(* IEC 61131-3 sources: AutomationStudio/BramaWjazdowa, 3 files *)

(* ---- Types.typ ---- *)
TYPE
	OperatorTyp : STRUCT
		diStart : BOOL;
		diStop : BOOL:= TRUE;
		diEStop : BOOL := TRUE;
		diKasujAwaria: BOOL; (*Przycisk kasowania awarii*)
		doSystemAktywny: BOOL; (*Lampka systemu aktywny*)
		doAwaria : BOOL; (*Lampka Awaria*)
		diGateOpen : BOOL;
		diGateClose : BOOL;
		Pilot : PilotTyp;
	END_STRUCT;

	PilotTyp : STRUCT
		diGateOpen : BOOL;
		diGateClose : BOOL;
		diEStop : BOOL := TRUE;
	END_STRUCT;

	GateTyp : STRUCT
		diSafetySensor : BOOL := TRUE;
		diGateClosed : BOOL:= TRUE;
		diGateOpened : BOOL:= TRUE;
		diTemperature : BOOL := TRUE;
		doOpenGate : BOOL;
		doCloseGate : BOOL;
		doLampa : BOOL;
	END_STRUCT;

	SystemTyp : STRUCT
		Operator : OperatorTyp;
		Gate : GateTyp;
	END_STRUCT;

END_TYPE

(* ---- Main.st ---- *)
PROGRAM _INIT
	(* Insert code here *)

END_PROGRAM

PROGRAM _CYCLIC
	(*Rozruch systemu*)
	Mechanizm[0].Operator.doSystemAktywny:=(Mechanizm[0].Operator.diStart OR Mechanizm[0].Operator.doSystemAktywny) AND
	Mechanizm[0].Operator.diStop AND Mechanizm[0].Operator.diEStop AND NOT(Mechanizm[0].Operator.doAwaria);

	(*Mechanizm otwierania bramy*)

	Mechanizm[0].Gate.doOpenGate := (Mechanizm[0].Operator.diGateOpen OR Mechanizm[0].Operator.Pilot.diGateOpen)
	AND NOT(Mechanizm[0].Operator.doAwaria) AND Mechanizm[0].Gate.diTemperature
	AND Mechanizm[0].Gate.diGateOpened;

//	Mechanizm[0].Operator.diGateOpen:=Mechanizm[0].Gate.doOpenGate;

	(*Mechanizm zamykania bramy*)

	Mechanizm[0].Gate.doCloseGate := (Mechanizm[0].Operator.diGateClose OR Mechanizm[0].Operator.Pilot.diGateClose)
	AND NOT(Mechanizm[0].Operator.doAwaria) AND Mechanizm[0].Gate.diTemperature AND Mechanizm[0].Gate.diSafetySensor
	AND Mechanizm[0].Gate.diGateClosed;

//	Mechanizm[0].Operator.diGateClose:=Mechanizm[0].Gate.doCloseGate;

	(*Diagnostyka*)
	Mechanizm[0].Operator.doAwaria := NOT(Mechanizm[0].Gate.diTemperature AND Mechanizm[0].Gate.diSafetySensor)
	OR (Mechanizm[0].Operator.doAwaria AND NOT(Mechanizm[0].Operator.diKasujAwaria))
	OR NOT(Mechanizm[0].Gate.diGateClosed OR Mechanizm[0].Gate.diGateOpened);

	ZegarTON[0].IN:=ZegarTOF[0].Q;
	ZegarTON[0].PT:= T#1000ms;
	ZegarTON[0]();

	ZegarTOF[0].IN:= NOT(ZegarTON[0].Q);
	ZegarTOF[0].PT:= T#1000ms;
	ZegarTOF[0]();

	Mechanizm[0].Gate.doLampa:= (Mechanizm[0].Operator.diGateOpen OR Mechanizm[0].Operator.diGateClose) AND ZegarTON[0].Q;

END_PROGRAM

PROGRAM _EXIT
	(* Insert code here *)

END_PROGRAM

(* ---- Variables.var ---- *)
VAR

	Mechanizm : ARRAY[0..1] OF SystemTyp;
	ZegarTON : ARRAY[0..1] OF TON;
	ZegarTOF : ARRAY[0..1] OF TOF;
END_VAR
